# EPICS StreamDevice protocol: ioc/rosApp/Db/ros.proto
ExtraInput = Ignore;
ReplyTimeout = 100;
#Terminator = LF;
#
getInput {
        #out "%(\$2:IN\$1:Units_RBV.VAL)s","RDG? ","%(\$2:OUT\$1:Cntrl_RBV.VAL)s";
        in "%(\$1.VAL)s";
    }
setOutput {
        out "%(\$1.VAL)s";
    }
